TYPE ST_Fan_ip :
STRUCT
	OnOffCmd 	AT%I* : BOOL;
	SpeedSp		AT%I* : INT;
END_STRUCT
END_TYPE

(* stored: Version 1.1.0.1, ProductVersion 3.1.4024.12
   DUT ST_Fan_ip: Id {630b47be-a342-4741-8403-f00638dfcdbe} *)
